Staubli VAL3: Float_Edit.pgx

public program Float_Edit(num& x_nData, num x_nX, num x_nY)
  local num l_nKey
  local num l_nNum
  local num l_nOri
begin
  //说明
  //对于数字的修改
  //使用get来实现对数字的修改


  //参数判断
  x_nX=min(max(0,x_nX),39)
  x_nY=min(max(0,x_nY),13)
  //x_nLength=min(max(getDisplayLen("")+1,x_nLength),39)
  setTextMode(0)
  //把字符串给打印出来
  gotoxy(x_nX,x_nY)
  l_nNum=x_nData
  put(left("                       ",nPanelWidthX-x_nX+nPanelLTopX+1))
  gotoxy(x_nX,x_nY)
  setTextMode(0)
  wait(get(l_nNum)==270)
  x_nData=l_nNum

end
